FUNCTION "bioBitSum" : VOID
TITLE = Count TRUE Bits
{ S7_Optimized_Access := 'TRUE' }
AUTHOR : Woermann
VERSION : 0.2
// -- Woermann Automation --
// Date: 2020-07-05
// Description:
// Count the number of TRUE Bits in a given Word (16 Bit)
// Using Brian Kernighan's C algorithm (v &= v - 1), only going through as many iterations as there are TRUE bits
// -- Inputs --
// InWord: Input word of wich the bits that are TRUE should be counted
// -- Outputs --
// OutByte: Result of counted TRUE Bits (Range is 0 to 16)


	VAR_INPUT
		InWord : WORD ;	// Input Word with Bits to be counted
	END_VAR

	VAR_OUTPUT
		OutByte : BYTE ;	// Output Byte (Counted Bits Result)
	END_VAR

BEGIN
	NETWORK
	TITLE = Count TRUE Bits

		L     0;
		T     #OutByte;
		L     #InWord;
		PUSH  ;
	L001: AW    ;
		T     #InWord;
		L     0;
		==D   ;
		BEC   ;
		L     #OutByte;
		INC   1;
		T     #OutByte;
		L     #InWord;
		PUSH  ;
		LOOP  L001;

END_FUNCTION

